// TIA Portal V21 export
DATA_BLOCK "DELTA D"   // DB183
{ S7_Optimized_Access := 'FALSE' }
   VAR
      TA : Real := 122.9;
      TB : Real := 121.0;
      Z : Real := 10.0;
      RATE : Real := 0.1900001;
      LEATHALTY : Real := 1.548817;
      "DELTA T" : Int := 15;
      F0 : Real := 13.06446;
      "MIN DRAIN" : Real := 51.8;
      "MAX DRAIN" : Real := 123.2;
      "MIN T1" : Real := 85.7;
      "MAX T1" : Real := 123.8;
      "MIN T2" : Real := 44.5;
      "MAX T2" : Real := 124.3;
      "MIN T3" : Real := 43.1;
      "MAX T3" : Real := 124.2;
      "MIN T4" : Real := 85.8;
      "MAX T4" : Real := 124.0;
      "MIN T5" : Real := 0.0;
      "MAX T5" : Real := 0.0;
      HEAD : String[80] := '$L$R                T1     T2     T3     T4      T5  ';   // 17,24,31,38,46
      "MIN TEMP" : String[80] := '$L$R  MIN TEMP  :                                                            ';   // 14
      "MAX TEMP" : String[80] := '$L$R  MAX TEMP  :                                                           ';   // 14
      "F ZERO" : String[80] := '$L$R  F0 VALUE  :                                                            ';   // 14
      "MIN F0" : String[80] := '$L$RTOTAL MINIMUM F0 VALUE ACHIEVED DURING CYLCE  :           ';   // 48
      "PRINT LINE" : String[80] := '   ';
      BIT : Array[0..10] of Bool;
      F1 : Real := 23.23226;
      F2 : Real := 27.93129;
      F3 : Real := 30.62606;
      F4 : Real := 30.62606;
      F5 : Real := 29.24768;
      "DEL TA" : Array[0..5] of Real;
      "DEL RATE" : Array[0..5] of Real;
      "DEL LEATH" : Array[0..5] of Real;
      dummy : Array[0..5] of Real;
   END_VAR
BEGIN
   BIT[0..10] := FALSE;
   "DEL TA"[0] := 123.7;
   "DEL TA"[1..2] := 124.1;
   "DEL TA"[3] := 123.9;
   "DEL TA"[4..5] := 0.0;
   "DEL RATE"[0] := 0.2699997;
   "DEL RATE"[1..2] := 0.3099999;
   "DEL RATE"[3] := 0.2900001;
   "DEL RATE"[4..5] := 0.0;
   "DEL LEATH"[0] := 1.862086;
   "DEL LEATH"[1..2] := 2.041737;
   "DEL LEATH"[3] := 1.949845;
   "DEL LEATH"[4..5] := 0.0;
END_DATA_BLOCK
